FUNCTION_BLOCK Manual
VAR
	Counter: CTUD;
	MotorTable: Motor;
	MotorBelt: Motor;
END_VAR

Counter();

gvl.PistonInputBackwards := TRUE;
gvl.PistonInputForward := FALSE;

gvl.MotorTableMove := FALSE;

gvl.PistonPress := FALSE;

gvl.PistonOutputBackwards := TRUE;
gvl.PistonOutputForward := FALSE;

gvl.MotorBeltMove := FALSE;
IF (gvl.ButtonBLT AND Counter.CV > 0) THEN
	Counter.CD := TRUE;
ELSE
	Counter.CD := FALSE;
END_IF


IF (gvl.ButtonBRT AND Counter.CV < 4) THEN
	Counter.CU := TRUE;
ELSE
	Counter.CU := FALSE;
END_IF

IF Counter.CV = 0 THEN
	IF gvl.ButtonBLB THEN
		gvl.PistonInputBackwards := FALSE;
		gvl.PistonInputForward := TRUE;
	ELSE
		gvl.PistonInputBackwards := TRUE;
		gvl.PistonInputForward := FALSE;
	END_IF
	
ELSIF Counter.CV = 1 THEN
	MotorTable(
		Forwards := gvl.ButtonBRB,
		Backwards := gvl.ButtonBLB,
		blockTime := T#0.5S,
		Active => gvl.MotorTableMove,
		Direction => gvl.MotorTableDirection
	);	
	
ELSIF Counter.CV = 2 THEN
	IF gvl.ButtonBLB THEN
		gvl.PistonPress := TRUE;
	ELSE
		gvl.PistonPress := FALSE;
	END_IF
	
ELSIF Counter.CV = 3 THEN
	IF gvl.ButtonBLB THEN
		gvl.PistonOutputBackwards := FALSE;
		gvl.PistonOutputForward := TRUE;
	ELSE
		gvl.PistonOutputBackwards := TRUE;
		gvl.PistonOutputForward := FALSE;
	END_IF
	
ELSIF Counter.CV = 4 THEN
	MotorBelt(
		Forwards := gvl.ButtonBRB,
		Backwards := gvl.ButtonBLB,
		blockTime := T#0.5S,
		Active => gvl.MotorBeltMove,
		Direction => gvl.MotorBeltDirection
	);
END_IF

END_FUNCTION_BLOCK

(* stored: Version 1.1.0.1, ProductVersion 3.1.4024.12
   POU Manual: Id {0ada9505-5641-4978-b97a-e28652d1bb28}, SpecialFunc None *)
